TYPE MaterialStorage :
STRUCT
	slots : ARRAY[0..GVL.maxQueue] OF STRING;
	units : ARRAY[0..GVL.maxQueue] OF INT;
END_STRUCT
END_TYPE

(* stored: Version 1.1.0.1, ProductVersion 3.1.4024.11
   DUT MaterialStorage: Id {590f9ee7-a84c-4ed6-8a24-e07398726f61} *)
